// TIA Portal project "Seviye ve Sıcaklık Kontrol" (V17)

(* hardware
DEVICE "S7-1500/ET200MP station_1"  S7-1500 station
   slot 0: "Rail_0"  Rack  6ES7 590-1***0-0AA0
   slot 1: "PLC_1"  CPU 1511C-1 PN  6ES7 511-1CK00-0AB0  V2.9
      slot 3: "CPU display_1"  6ES7591-1AA00-0AA0
      slot 32768: "PROFINET interface_1"  X1
         slot 32769: "Port_1"  X1 P1
         slot 32770: "Port_2"  X1 P2
      slot 34817: "Virtual CP interface port_1"  Virtual CP interface port  Virtual CP interface port
DEVICE "HMI_1"  TP700 Comfort
   slot 0: "HMI_1"  TP700 Comfort  6AV2 124-0GC01-0AX0  17.0.0.0
   slot 1: "HMI_RT_1"  TP700 Comfort  6AV2 124-0GC01-0AX0  17.0.0.0
   slot 5: "HMI_1.IE_CP_1"  PROFINET Interface  17.0.0.0
      slot 1: "PROFINET Interface_1"  PROFINET Interface
         slot 1: "Port_1"  Port
         slot 2: "Port_2"  Port
   slot 7: "HMI_1.MPI/DP_CP_1"  MPI/DP Interface  17.0.0.0
*)

// ===== PLC "PLC_1"  CPU 1511C-1 PN =====

VAR_GLOBAL   // PLC tag table "Default tag table"
   "Otomatik Çalışma Aktif" AT %M1.0 : Bool;
   "Seviye Set Değer" AT %MD60 : Real;
   "Sıcaklık Set Değer" AT %MD40 : Real;
   "Seviye_OK" AT %M1.3 : Bool;
   "Taşma_Sensörü" AT %MD116 : Real;
   "Tag_1" AT %MD132 : DWord;
   "Anlık Seviye" AT %MD30 : DWord;
   "Anlık Sıcaklık Değeri" AT %MD46 : DWord;
   "Sistem Sıcaklık Değeri" AT %MD62 : DWord;
   "Sistem Seviye Değeri" AT %MD78 : DWord;
   "Manuel Çalışma Aktif" AT %M1.6 : Bool;
   "Sıcaklık_OK" AT %M1.1 : Bool;
   "Kullanıcıdan Alınan Zaman Değeri (Dakika)" AT %MD8 : Time;
   "Timer Zaman Değeri" AT %MD16 : Time;
   "Sistem Tamamlandı" AT %M1.2 : Bool;
   "Sistem Aşırı Sıcak" AT %M1.4 : Bool;
   "Sistem Aşırı Seviye" AT %M1.5 : Bool;
END_VAR

VAR_GLOBAL   // PLC tag table "Dijital Outputlar"
   "Pompa Motoru" AT %Q4.0 : Bool;
   "Isıtıcı" AT %Q4.1 : Bool;
   "Karıştırma Motoru" AT %Q4.2 : Bool;
   "System_OK Sesli Uyarı Sireni" AT %Q4.3 : Bool;
   "System OK Lamba" AT %Q4.4 : Bool;
   "Uyarı Kırmızı Lamba" AT %Q4.5 : Bool;
   "Uyarı Sireni" AT %Q4.6 : Bool;
   "Pompa Motoru Sürücüsü" AT %Q4.7 : Bool;
   "Karıştırma Motoru Sürücüsü" AT %Q5.0 : Bool;
END_VAR

VAR_GLOBAL   // PLC tag table "Analog Output"
   "Pompa Motoru Sürücü" AT %QW0 : Int;
   "SCR" AT %QW2 : Int;
END_VAR

VAR_GLOBAL   // PLC tag table "Dijital Inputlar"
   "Oto Start" AT %I10.0 : Bool;
   "Manuel Start Butonu" AT %I10.1 : Bool;
   "Stop Butonu" AT %I10.2 : Bool;
   "Acil Stop Butonu" AT %I10.3 : Bool;
   "Pompa Motoru Manuel Çalışma" AT %I10.4 : Bool;
   "Isıtıcı Manuel Çalışma" AT %I10.5 : Bool;
   "Karıştırma Motoru Manuel Çalıştırma Butonu" AT %I10.6 : Bool;
END_VAR

VAR_GLOBAL   // PLC tag table "Analog Inputlar"
   "Seviye Ölçer Sensörü" AT %IW0 : Int;
   "Pt100" AT %IW2 : Int;
   "Sistem Sıcaklık Sensörü" AT %IW4 : Word;
   "Taşma Sensörü" AT %IW6 : Word;
END_VAR

DATA_BLOCK "db_HMI"   // DB2
{ S7_Optimized_Access := 'TRUE' }
VERSION : 0.1
   VAR
      "Pompa Motoru Manuel Çalışma" : Bool;
      "Isıtıcı Manuel Çalışma" : Bool;
      "Karıştırma Motoru Manuel Çalıştırma" : Bool;
      "Seviye PID Manuel Çalışma" : Bool;
      "Sıcaklık PID Manuel Çalışma" : Bool;
      "HMI Oto Start" : Bool;
      "HMI Manuel Start" : Bool;
   END_VAR
BEGIN
END_DATA_BLOCK

DATA_BLOCK "db_Alarmlar"   // DB4
{ S7_Optimized_Access := 'FALSE' }
VERSION : 0.1
   VAR
      "Stop Butonuna Basıldı" : Bool;
      "Acil Stop Butonu Basılı" : Bool;
      "Sistem Aşırı Sıcak Değeri" : Bool;
      "Sistem Aşırı Seviye Değeri" : Bool;
      "Seviye Ölçer Sensörü Kablosu Koptu" : Bool;
      "Pt100 Sensörü Kablosu Koptu" : Bool;
      "Taşma Sensörü Kablosu Koptu" : Bool;
      "Sistem Sıcaklık Sensörü Kablosu Koptu" : Bool;
   END_VAR
BEGIN
END_DATA_BLOCK

// folder: System blocks/Program resources

DATA_BLOCK "Zamanlayıcı"   // DB5
{ S7_Optimized_Access := 'TRUE' }
AUTHOR : Simatic
FAMILY : IEC
NAME : IEC_TMR
VERSION : 1.0
// stored: InstanceOfName IEC_TIMER
"IEC_TIMER"
BEGIN
END_DATA_BLOCK

// folder: (top level)

FUNCTION "HMI Alarmlar" : Void   // FC1, LAD
{ S7_Optimized_Access := 'TRUE' }
VERSION : 0.1
BEGIN

REGION Network 1
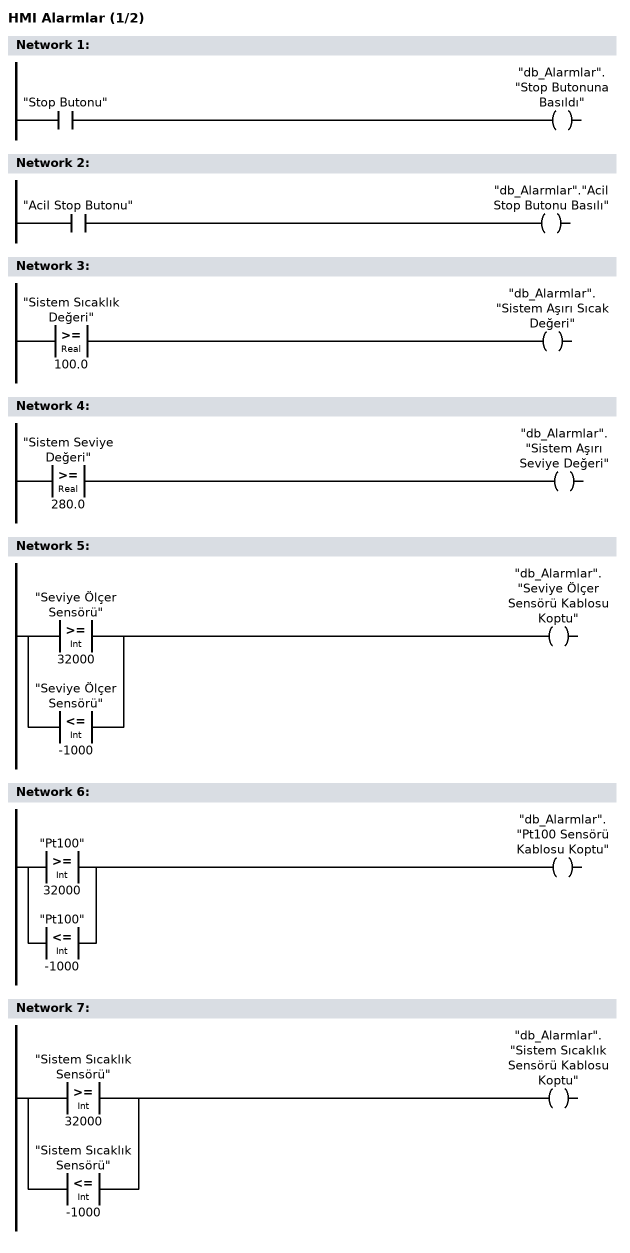
   RUNG wire#powerrail
      Contact( "Stop Butonu" )
      Coil( "db_Alarmlar"."Stop Butonuna Basıldı" )
   END_RUNG
   // the same network as SCL:
   "db_Alarmlar"."Stop Butonuna Basıldı" := "Stop Butonu";
END_REGION

REGION Network 2
   RUNG wire#powerrail
      Contact( "Acil Stop Butonu" )
      Coil( "db_Alarmlar"."Acil Stop Butonu Basılı" )
   END_RUNG
   // the same network as SCL:
   "db_Alarmlar"."Acil Stop Butonu Basılı" := "Acil Stop Butonu";
END_REGION

REGION Network 3
   RUNG wire#powerrail
      { S7_Templates := "SrcType := Real" } GE_Contact(in1 := "Sistem Sıcaklık Değeri", in2 := 100.0)
      Coil( "db_Alarmlar"."Sistem Aşırı Sıcak Değeri" )
   END_RUNG
   // the same network as SCL:
   "db_Alarmlar"."Sistem Aşırı Sıcak Değeri" := "Sistem Sıcaklık Değeri" >= 100.0;
END_REGION

REGION Network 4
   RUNG wire#powerrail
      { S7_Templates := "SrcType := Real" } GE_Contact(in1 := "Sistem Seviye Değeri", in2 := 280.0)
      Coil( "db_Alarmlar"."Sistem Aşırı Seviye Değeri" )
   END_RUNG
   // the same network as SCL:
   "db_Alarmlar"."Sistem Aşırı Seviye Değeri" := "Sistem Seviye Değeri" >= 280.0;
END_REGION

REGION Network 5
   RUNG wire#powerrail
      { S7_Templates := "SrcType := Int" } GE_Contact(in1 := "Seviye Ölçer Sensörü", in2 := 32000)
      wire#w1
      Coil( "db_Alarmlar"."Seviye Ölçer Sensörü Kablosu Koptu" )
   END_RUNG
   RUNG wire#powerrail
      { S7_Templates := "SrcType := Int" } LE_Contact(in1 := "Seviye Ölçer Sensörü", in2 := -1000)
   END_RUNG wire#w1
   // the same network as SCL:
   "db_Alarmlar"."Seviye Ölçer Sensörü Kablosu Koptu" := ("Seviye Ölçer Sensörü" >= 32000) OR ("Seviye Ölçer Sensörü" <= (-1000));
END_REGION

REGION Network 6
   RUNG wire#powerrail
      { S7_Templates := "SrcType := Int" } GE_Contact(in1 := "Pt100", in2 := 32000)
      wire#w1
      Coil( "db_Alarmlar"."Pt100 Sensörü Kablosu Koptu" )
   END_RUNG
   RUNG wire#powerrail
      { S7_Templates := "SrcType := Int" } LE_Contact(in1 := "Pt100", in2 := -1000)
   END_RUNG wire#w1
   // the same network as SCL:
   "db_Alarmlar"."Pt100 Sensörü Kablosu Koptu" := ("Pt100" >= 32000) OR ("Pt100" <= (-1000));
END_REGION

REGION Network 7
   RUNG wire#powerrail
      { S7_Templates := "SrcType := Int" } GE_Contact(in1 := "Sistem Sıcaklık Sensörü", in2 := 32000)
      wire#w1
      Coil( "db_Alarmlar"."Sistem Sıcaklık Sensörü Kablosu Koptu" )
   END_RUNG
   RUNG wire#powerrail
      { S7_Templates := "SrcType := Int" } LE_Contact(in1 := "Sistem Sıcaklık Sensörü", in2 := -1000)
   END_RUNG wire#w1
   // the same network as SCL:
   "db_Alarmlar"."Sistem Sıcaklık Sensörü Kablosu Koptu" := ("Sistem Sıcaklık Sensörü" >= 32000) OR ("Sistem Sıcaklık Sensörü" <= (-1000));
END_REGION

REGION Network 8
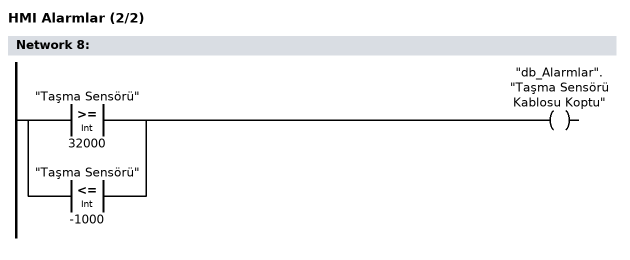
   RUNG wire#powerrail
      { S7_Templates := "SrcType := Int" } GE_Contact(in1 := "Taşma Sensörü", in2 := 32000)
      wire#w1
      Coil( "db_Alarmlar"."Taşma Sensörü Kablosu Koptu" )
   END_RUNG
   RUNG wire#powerrail
      { S7_Templates := "SrcType := Int" } LE_Contact(in1 := "Taşma Sensörü", in2 := -1000)
   END_RUNG wire#w1
   // the same network as SCL:
   "db_Alarmlar"."Taşma Sensörü Kablosu Koptu" := ("Taşma Sensörü" >= 32000) OR ("Taşma Sensörü" <= (-1000));
END_REGION
END_FUNCTION

FUNCTION "Manuel Çalışma" : Void   // FC2, LAD
{ S7_Optimized_Access := 'TRUE' }
VERSION : 0.1
BEGIN

REGION Network 1: Manuel Çalışma Modu
   // Manuel Start ile Merker biti aktif edilir.
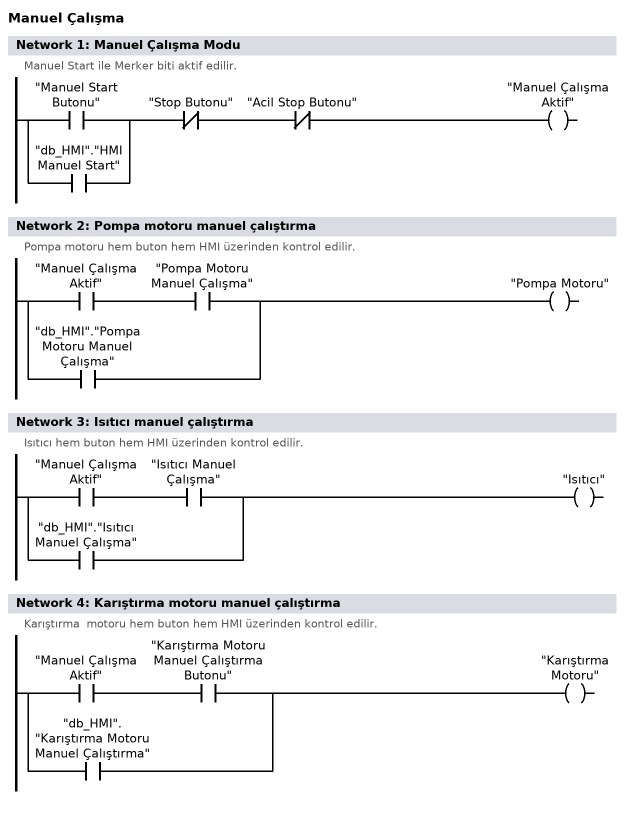
   RUNG wire#powerrail
      Contact( "Manuel Start Butonu" )
      wire#w1
      I_Contact( "Stop Butonu" )
      I_Contact( "Acil Stop Butonu" )
      Coil( "Manuel Çalışma Aktif" )
   END_RUNG
   RUNG wire#powerrail
      Contact( "db_HMI"."HMI Manuel Start" )
   END_RUNG wire#w1
   // the same network as SCL:
   "Manuel Çalışma Aktif" := ("Manuel Start Butonu" OR "db_HMI"."HMI Manuel Start") AND NOT "Stop Butonu" AND NOT "Acil Stop Butonu";
END_REGION

REGION Network 2: Pompa motoru manuel çalıştırma
   // Pompa motoru hem buton hem HMI üzerinden kontrol edilir.
   RUNG wire#powerrail
      Contact( "Manuel Çalışma Aktif" )
      Contact( "Pompa Motoru Manuel Çalışma" )
      wire#w1
      Coil( "Pompa Motoru" )
   END_RUNG
   RUNG wire#powerrail
      Contact( "db_HMI"."Pompa Motoru Manuel Çalışma" )
   END_RUNG wire#w1
   // the same network as SCL:
   "Pompa Motoru" := ("Manuel Çalışma Aktif" AND "Pompa Motoru Manuel Çalışma") OR "db_HMI"."Pompa Motoru Manuel Çalışma";
END_REGION

REGION Network 3: Isıtıcı manuel çalıştırma
   // Isıtıcı hem buton hem HMI üzerinden kontrol edilir.
   RUNG wire#powerrail
      Contact( "Manuel Çalışma Aktif" )
      Contact( "Isıtıcı Manuel Çalışma" )
      wire#w1
      Coil( "Isıtıcı" )
   END_RUNG
   RUNG wire#powerrail
      Contact( "db_HMI"."Isıtıcı Manuel Çalışma" )
   END_RUNG wire#w1
   // the same network as SCL:
   "Isıtıcı" := ("Manuel Çalışma Aktif" AND "Isıtıcı Manuel Çalışma") OR "db_HMI"."Isıtıcı Manuel Çalışma";
END_REGION

REGION Network 4: Karıştırma motoru manuel çalıştırma
   // Karıştırma  motoru hem buton hem HMI üzerinden kontrol edilir.
   RUNG wire#powerrail
      Contact( "Manuel Çalışma Aktif" )
      Contact( "Karıştırma Motoru Manuel Çalıştırma Butonu" )
      wire#w1
      Coil( "Karıştırma Motoru" )
   END_RUNG
   RUNG wire#powerrail
      Contact( "db_HMI"."Karıştırma Motoru Manuel Çalıştırma" )
   END_RUNG wire#w1
   // the same network as SCL:
   "Karıştırma Motoru" := ("Manuel Çalışma Aktif" AND "Karıştırma Motoru Manuel Çalıştırma Butonu") OR "db_HMI"."Karıştırma Motoru Manuel Çalıştırma";
END_REGION
END_FUNCTION

FUNCTION "Otomatik Çalışma" : Void   // FC3, LAD
{ S7_Optimized_Access := 'TRUE' }
VERSION : 0.1
BEGIN

REGION Network 1: Başlangıç
   // Start butonuna basarak sistemi aktif ederiz. Sistem aktif bilgisini merker bitiyle bağlayıp diğer adımlarda rahatlıkla kullanılır.
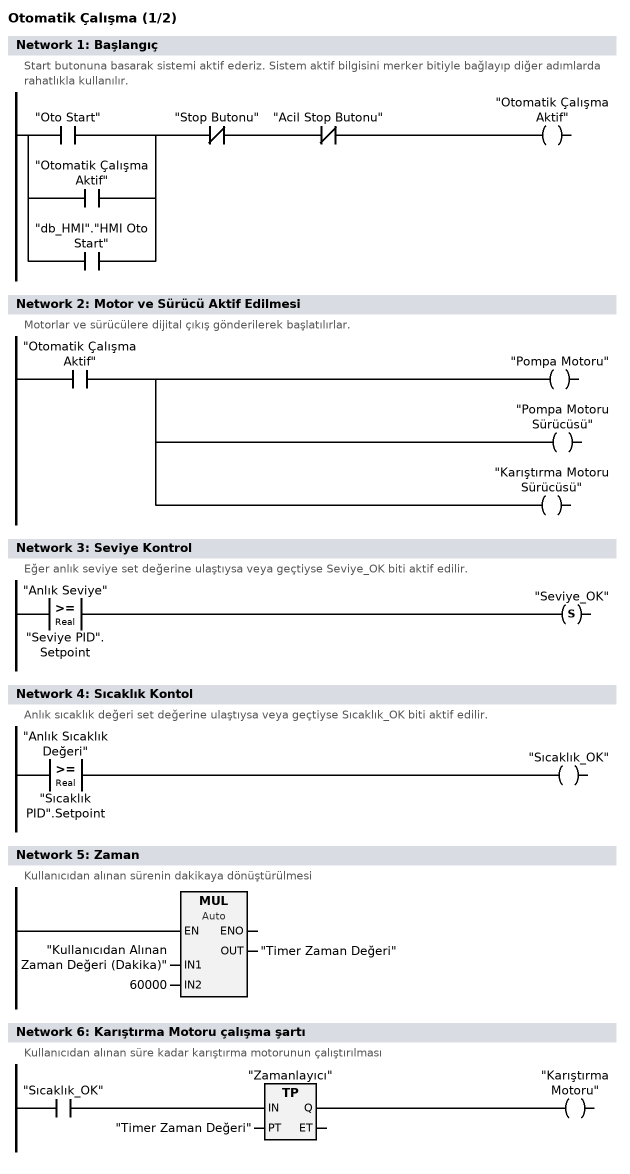
   RUNG wire#powerrail
      Contact( "Oto Start" )
      wire#w1
      I_Contact( "Stop Butonu" )
      I_Contact( "Acil Stop Butonu" )
      Coil( "Otomatik Çalışma Aktif" )
   END_RUNG
   RUNG wire#powerrail
      Contact( "Otomatik Çalışma Aktif" )
   END_RUNG wire#w1
   RUNG wire#powerrail
      Contact( "db_HMI"."HMI Oto Start" )
   END_RUNG wire#w1
   // the same network as SCL:
   "Otomatik Çalışma Aktif" := ("Oto Start" OR "Otomatik Çalışma Aktif" OR "db_HMI"."HMI Oto Start") AND NOT "Stop Butonu" AND NOT "Acil Stop Butonu";
END_REGION

REGION Network 2: Motor ve Sürücü Aktif Edilmesi
   // Motorlar ve sürücülere dijital çıkış gönderilerek başlatılırlar.
   RUNG wire#powerrail
      Contact( "Otomatik Çalışma Aktif" )
      wire#w1
      Coil( "Pompa Motoru" )
   END_RUNG
   RUNG wire#w1
      Coil( "Pompa Motoru Sürücüsü" )
   END_RUNG
   RUNG wire#w1
      Coil( "Karıştırma Motoru Sürücüsü" )
   END_RUNG
   // the same network as SCL:
   "Pompa Motoru" := "Otomatik Çalışma Aktif";
   "Pompa Motoru Sürücüsü" := "Otomatik Çalışma Aktif";
   "Karıştırma Motoru Sürücüsü" := "Otomatik Çalışma Aktif";
END_REGION

REGION Network 3: Seviye Kontrol
   // Eğer anlık seviye set değerine ulaştıysa veya geçtiyse Seviye_OK biti aktif edilir.
   RUNG wire#powerrail
      { S7_Templates := "SrcType := Real" } GE_Contact(in1 := "Anlık Seviye", in2 := "Seviye PID".Setpoint)
      S_Coil( "Seviye_OK" )
   END_RUNG
   // the same network as SCL:
   IF "Anlık Seviye" >= "Seviye PID".Setpoint THEN "Seviye_OK" := TRUE; END_IF;
END_REGION

REGION Network 4: Sıcaklık Kontol
   // Anlık sıcaklık değeri set değerine ulaştıysa veya geçtiyse Sıcaklık_OK biti aktif edilir.
   RUNG wire#powerrail
      { S7_Templates := "SrcType := Real" } GE_Contact(in1 := "Anlık Sıcaklık Değeri", in2 := "Sıcaklık PID".Setpoint)
      Coil( "Sıcaklık_OK" )
   END_RUNG
   // the same network as SCL:
   "Sıcaklık_OK" := "Anlık Sıcaklık Değeri" >= "Sıcaklık PID".Setpoint;
END_REGION

REGION Network 5: Zaman
   // Kullanıcıdan alınan sürenin dakikaya dönüştürülmesi
   RUNG wire#powerrail
      Mul(in1 := "Kullanıcıdan Alınan Zaman Değeri (Dakika)", in2 := 60000, out => "Timer Zaman Değeri")
   END_RUNG
   // the same network as SCL:
   "Timer Zaman Değeri" := "Kullanıcıdan Alınan Zaman Değeri (Dakika)" * 60000;
END_REGION

REGION Network 6: Karıştırma Motoru çalışma şartı
   // Kullanıcıdan alınan süre kadar karıştırma motorunun çalıştırılması
   "Zamanlayıcı".TP(IN := "Sıcaklık_OK", PT := "Timer Zaman Değeri");
   "Karıştırma Motoru" := "Zamanlayıcı".Q;
END_REGION

REGION Network 7: Sistemin tamamlanması
   // Seviye set değerine ulaştıysa, Sıcaklık set değerine ulaştıysa ve karıştıma motoru istenilen zaman aralığında çalıştıysa sistem tamamlandı demektir.
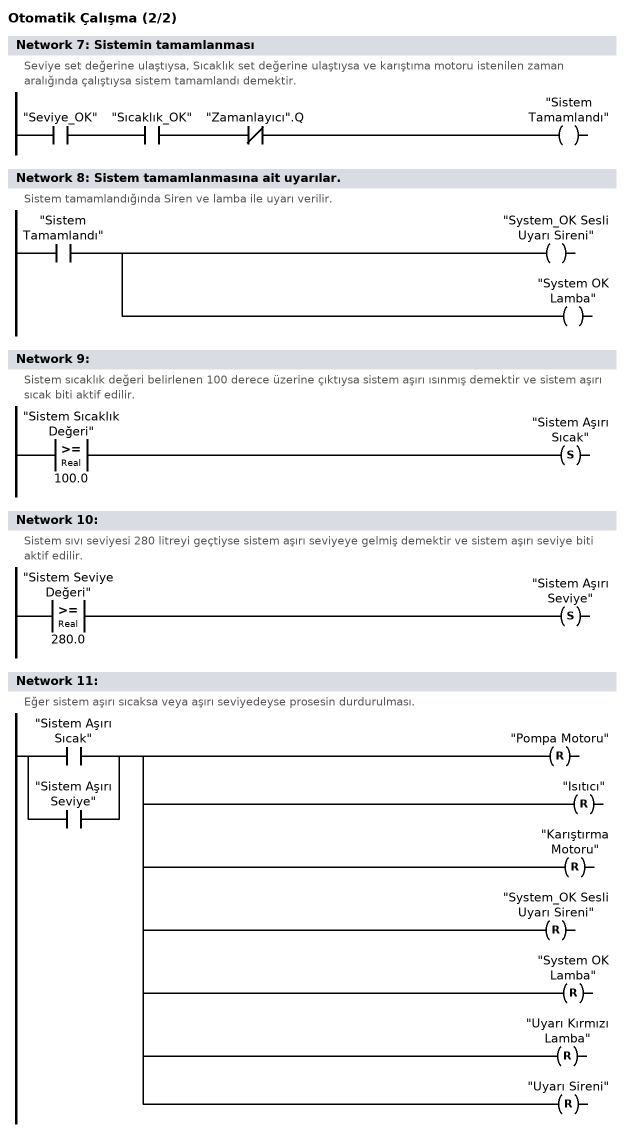
   RUNG wire#powerrail
      Contact( "Seviye_OK" )
      Contact( "Sıcaklık_OK" )
      I_Contact( "Zamanlayıcı".Q )
      Coil( "Sistem Tamamlandı" )
   END_RUNG
   // the same network as SCL:
   "Sistem Tamamlandı" := "Seviye_OK" AND "Sıcaklık_OK" AND NOT "Zamanlayıcı".Q;
END_REGION

REGION Network 8: Sistem tamamlanmasına ait uyarılar.
   // Sistem tamamlandığında Siren ve lamba ile uyarı verilir.
   RUNG wire#powerrail
      Contact( "Sistem Tamamlandı" )
      wire#w1
      Coil( "System_OK Sesli Uyarı Sireni" )
   END_RUNG
   RUNG wire#w1
      Coil( "System OK Lamba" )
   END_RUNG
   // the same network as SCL:
   "System_OK Sesli Uyarı Sireni" := "Sistem Tamamlandı";
   "System OK Lamba" := "Sistem Tamamlandı";
END_REGION

REGION Network 9
   // Sistem sıcaklık değeri belirlenen 100 derece üzerine çıktıysa sistem aşırı ısınmış demektir ve sistem aşırı sıcak biti aktif edilir.
   RUNG wire#powerrail
      { S7_Templates := "SrcType := Real" } GE_Contact(in1 := "Sistem Sıcaklık Değeri", in2 := 100.0)
      S_Coil( "Sistem Aşırı Sıcak" )
   END_RUNG
   // the same network as SCL:
   IF "Sistem Sıcaklık Değeri" >= 100.0 THEN "Sistem Aşırı Sıcak" := TRUE; END_IF;
END_REGION

REGION Network 10
   // Sistem sıvı seviyesi 280 litreyi geçtiyse sistem aşırı seviyeye gelmiş demektir ve sistem aşırı seviye biti aktif edilir.
   RUNG wire#powerrail
      { S7_Templates := "SrcType := Real" } GE_Contact(in1 := "Sistem Seviye Değeri", in2 := 280.0)
      S_Coil( "Sistem Aşırı Seviye" )
   END_RUNG
   // the same network as SCL:
   IF "Sistem Seviye Değeri" >= 280.0 THEN "Sistem Aşırı Seviye" := TRUE; END_IF;
END_REGION

REGION Network 11
   // Eğer sistem aşırı sıcaksa veya aşırı seviyedeyse prosesin durdurulması.
   RUNG wire#powerrail
      Contact( "Sistem Aşırı Sıcak" )
      wire#w1
      R_Coil( "Pompa Motoru" )
   END_RUNG
   RUNG wire#powerrail
      Contact( "Sistem Aşırı Seviye" )
   END_RUNG wire#w1
   RUNG wire#w1
      R_Coil( "Isıtıcı" )
   END_RUNG
   RUNG wire#w1
      R_Coil( "Karıştırma Motoru" )
   END_RUNG
   RUNG wire#w1
      R_Coil( "System_OK Sesli Uyarı Sireni" )
   END_RUNG
   RUNG wire#w1
      R_Coil( "System OK Lamba" )
   END_RUNG
   RUNG wire#w1
      R_Coil( "Uyarı Kırmızı Lamba" )
   END_RUNG
   RUNG wire#w1
      R_Coil( "Uyarı Sireni" )
   END_RUNG
   // the same network as SCL:
   IF "Sistem Aşırı Sıcak" OR "Sistem Aşırı Seviye" THEN
       "Pompa Motoru" := FALSE;
       "Isıtıcı" := FALSE;
       "Karıştırma Motoru" := FALSE;
       "System_OK Sesli Uyarı Sireni" := FALSE;
       "System OK Lamba" := FALSE;
       "Uyarı Kırmızı Lamba" := FALSE;
       "Uyarı Sireni" := FALSE;
   END_IF;
END_REGION
END_FUNCTION

ORGANIZATION_BLOCK "Main"   // OB1, LAD, ProgramCycle
TITLE = "Main Program Sweep (Cycle)"
{ S7_Optimized_Access := 'TRUE' }
VERSION : 0.1
   VAR_INPUT
      Initial_Call : Bool;   // Initial call of this OB
      Remanence : Bool;   // =True, if remanent data are available
   END_VAR
   VAR_TEMP
      NORMX_Out : Real;
      NORMX_Out_1 : Real;
      NORMX_Out_2 : Real;
      NORMX_Out_3 : Real;
   END_VAR
BEGIN

REGION Network 1: Seviye Ölçer Sensörü Normalizasyon ve Skala İşlemi
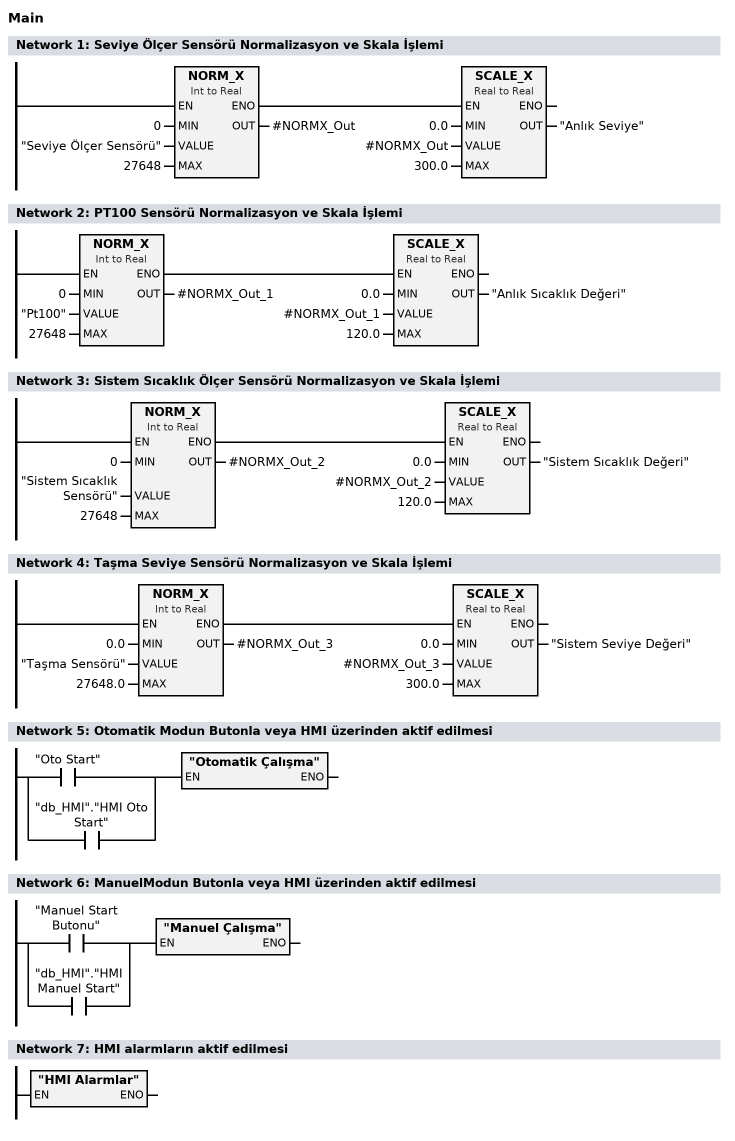
   RUNG wire#powerrail
      { S7_Templates := "[SrcType := Int, DestType := Real]" } Normalize(min := 0, value := "Seviye Ölçer Sensörü", max := 27648, out => #NORMX_Out)
      { S7_Templates := "[SrcType := Real, DestType := Real]" } Scale(min := 0.0, value := #NORMX_Out, max := 300.0, out => "Anlık Seviye")
   END_RUNG
   // the same network as SCL:
   #NORMX_Out := NORM_X(MIN := 0, VALUE := "Seviye Ölçer Sensörü", MAX := 27648);
   "Anlık Seviye" := SCALE_X(MIN := 0.0, VALUE := #NORMX_Out, MAX := 300.0);
END_REGION

REGION Network 2: PT100 Sensörü Normalizasyon ve Skala İşlemi
   RUNG wire#powerrail
      { S7_Templates := "[SrcType := Int, DestType := Real]" } Normalize(min := 0, value := "Pt100", max := 27648, out => #NORMX_Out_1)
      { S7_Templates := "[SrcType := Real, DestType := Real]" } Scale(min := 0.0, value := #NORMX_Out_1, max := 120.0, out => "Anlık Sıcaklık Değeri")
   END_RUNG
   // the same network as SCL:
   #NORMX_Out_1 := NORM_X(MIN := 0, VALUE := "Pt100", MAX := 27648);
   "Anlık Sıcaklık Değeri" := SCALE_X(MIN := 0.0, VALUE := #NORMX_Out_1, MAX := 120.0);
END_REGION

REGION Network 3: Sistem Sıcaklık Ölçer Sensörü Normalizasyon ve Skala İşlemi
   RUNG wire#powerrail
      { S7_Templates := "[SrcType := Int, DestType := Real]" } Normalize(min := 0, value := "Sistem Sıcaklık Sensörü", max := 27648, out => #NORMX_Out_2)
      { S7_Templates := "[SrcType := Real, DestType := Real]" } Scale(min := 0.0, value := #NORMX_Out_2, max := 120.0, out => "Sistem Sıcaklık Değeri")
   END_RUNG
   // the same network as SCL:
   #NORMX_Out_2 := NORM_X(MIN := 0, VALUE := "Sistem Sıcaklık Sensörü", MAX := 27648);
   "Sistem Sıcaklık Değeri" := SCALE_X(MIN := 0.0, VALUE := #NORMX_Out_2, MAX := 120.0);
END_REGION

REGION Network 4: Taşma Seviye Sensörü Normalizasyon ve Skala İşlemi
   RUNG wire#powerrail
      { S7_Templates := "[SrcType := Int, DestType := Real]" } Normalize(min := 0.0, value := "Taşma Sensörü", max := 27648.0, out => #NORMX_Out_3)
      { S7_Templates := "[SrcType := Real, DestType := Real]" } Scale(min := 0.0, value := #NORMX_Out_3, max := 300.0, out => "Sistem Seviye Değeri")
   END_RUNG
   // the same network as SCL:
   #NORMX_Out_3 := NORM_X(MIN := 0.0, VALUE := "Taşma Sensörü", MAX := 27648.0);
   "Sistem Seviye Değeri" := SCALE_X(MIN := 0.0, VALUE := #NORMX_Out_3, MAX := 300.0);
END_REGION

REGION Network 5: Otomatik Modun Butonla veya HMI üzerinden aktif edilmesi
   RUNG wire#powerrail
      Contact( "Oto Start" )
      wire#w1
      "Otomatik Çalışma"()
   END_RUNG
   RUNG wire#powerrail
      Contact( "db_HMI"."HMI Oto Start" )
   END_RUNG wire#w1
   // the same network as SCL:
   IF "Oto Start" OR "db_HMI"."HMI Oto Start" THEN "Otomatik Çalışma"(); END_IF;
END_REGION

REGION Network 6: ManuelModun Butonla veya HMI üzerinden aktif edilmesi
   RUNG wire#powerrail
      Contact( "Manuel Start Butonu" )
      wire#w1
      "Manuel Çalışma"()
   END_RUNG
   RUNG wire#powerrail
      Contact( "db_HMI"."HMI Manuel Start" )
   END_RUNG wire#w1
   // the same network as SCL:
   IF "Manuel Start Butonu" OR "db_HMI"."HMI Manuel Start" THEN "Manuel Çalışma"(); END_IF;
END_REGION

REGION Network 7: HMI alarmların aktif edilmesi
   RUNG wire#powerrail
      "HMI Alarmlar"()
   END_RUNG
   // the same network as SCL:
   "HMI Alarmlar"();
END_REGION
END_ORGANIZATION_BLOCK

ORGANIZATION_BLOCK "Seviye PID Kontrol"   // OB30, LAD, CyclicInterrupt
{ S7_Optimized_Access := 'TRUE' }
VERSION : 0.1
   VAR_INPUT
      Initial_Call : Bool;   // Initial call of this OB
      Event_Count : Int;   // Events discarded
   END_VAR
BEGIN

REGION Network 1: Seviye PID bloğunun aktif edilmesi
   // Hem otomatik hem manuel modda aktif edilebilir. Setpoint kısmına hafıza bitiatayarak HMI üzerinden değer girilebilir. Input_PER kısmını analog input girilir. Output_PER kısmına analog çıkış atanır. Seviye kontrolü için seviye bilgisi veren, analog seviye ölçer sensörünü Input_PER kısmına girip seviye değeri alınır. Daha sonra çıkışa motoru hız kontrollü çalıştırmak için sürücü atanır. Sürücü frekans artırıp azaltarak sürücüyü hız kontrolle çalıştırır.
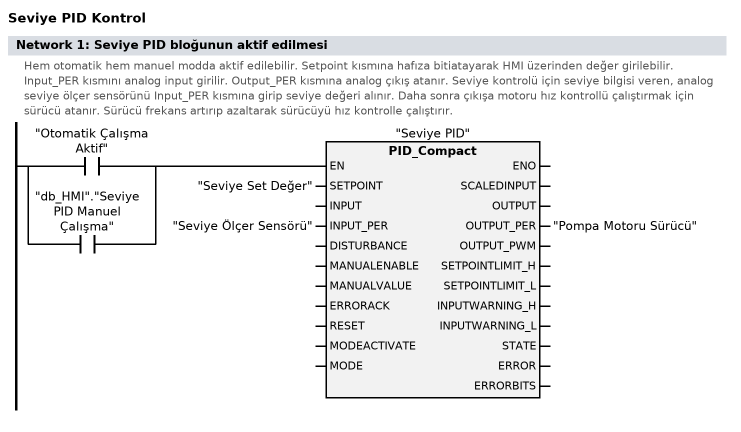
   IF "Otomatik Çalışma Aktif" OR "db_HMI"."Seviye PID Manuel Çalışma" THEN
       "Seviye PID"(Setpoint := "Seviye Set Değer",   // PID_Compact
                    Input_PER := "Seviye Ölçer Sensörü",
                    Output_PER => "Pompa Motoru Sürücü");
   END_IF;
END_REGION
END_ORGANIZATION_BLOCK

ORGANIZATION_BLOCK "Sıcaklık PID Kontrol"   // OB31, LAD, CyclicInterrupt
{ S7_Optimized_Access := 'TRUE' }
VERSION : 0.1
   VAR_INPUT
      Initial_Call : Bool;   // Initial call of this OB
      Event_Count : Int;   // Events discarded
   END_VAR
BEGIN

REGION Network 1: Sıcaklık PID Bloğunun Aktif Edilmesi
   // Setpoint kısmına hafıza bitiatayarak HMI üzerinden değer girilebilir. Input_PER kısmını analog input girilir. Output_PER kısmına analog çıkış atanır. Sıcalık kontrolü için sıcaklık bilgisi veren, pt100 sensörünü Input_PER kısmına girip seviye değeri alınır. Daha sonra çıkışa ısıtıcıyı kademeli olarak  çalıştırmak için scr cihazı atanır.
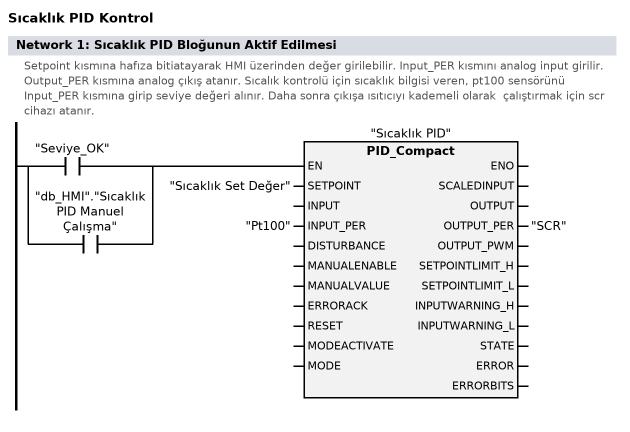
   IF "Seviye_OK" OR "db_HMI"."Sıcaklık PID Manuel Çalışma" THEN
       "Sıcaklık PID"(Setpoint := "Sıcaklık Set Değer", Input_PER := "Pt100", Output_PER => "SCR");   // PID_Compact
   END_IF;
END_REGION
END_ORGANIZATION_BLOCK

(* ===== HMI "HMI_RT_1" =====
system functions are stored by id; their names below are inferred from use
connection "HMI_Connection_1": ETHERNET, S7_1500_OMS

HMI tags "Default tag table"
   "Tag_ScreenNumber" : UInt, internal
   "db_HMI_HMI Oto Start" : Bool = PLC db_HMI."HMI Oto Start", 1 s
   "db_HMI_HMI Manuel Start" : Bool = PLC db_HMI."HMI Manuel Start", 1 s
   "Sistem Seviye Değeri" : DWord = PLC "Sistem Seviye Değeri" AT %MD78, 1 s
   "Sistem Sıcaklık Değeri" : DWord = PLC "Sistem Sıcaklık Değeri" AT %MD62, 1 s
   "Kullanıcıdan Alınan Zaman Değeri (Dakika)" : Time = PLC "Kullanıcıdan Alınan Zaman Değeri (Dakika)" AT %MD8, 1 s
   "db_HMI_Pompa Motoru Manuel Çalışma" : Bool = PLC db_HMI."Pompa Motoru Manuel Çalışma", 1 s
   "db_HMI_Isıtıcı Manuel Çalışma" : Bool = PLC db_HMI."Isıtıcı Manuel Çalışma", 1 s
   "db_HMI_Karıştırma Motoru Manuel Çalıştırma" : Bool = PLC db_HMI."Karıştırma Motoru Manuel Çalıştırma", 1 s
   "Pompa Motoru" : Bool = PLC "Pompa Motoru" AT %Q4.0, 1 s
   "Isıtıcı" : Bool = PLC Isıtıcı AT %Q4.1, 1 s
   "Karıştırma Motoru" : Bool = PLC "Karıştırma Motoru" AT %Q4.2, 1 s
   "Seviye Set Değer" : Real = PLC "Seviye Set Değer" AT %MD60, 1 s
   "Anlık Seviye" : DWord = PLC "Anlık Seviye" AT %MD30, 1 s
   "Seviye PID_Retain_CtrlParams_Ti" : Real = PLC "Seviye PID".Retain.CtrlParams.Ti, 1 s
   "Seviye PID_Retain_CtrlParams_Gain" : Real = PLC "Seviye PID".Retain.CtrlParams.Gain, 1 s
   "Seviye PID_Retain_CtrlParams_Td" : Real = PLC "Seviye PID".Retain.CtrlParams.Td, 1 s
   "Anlık Sıcaklık Değeri" : DWord = PLC "Anlık Sıcaklık Değeri" AT %MD46, 1 s
   "Sıcaklık Set Değer" : Real = PLC "Sıcaklık Set Değer" AT %MD40, 1 s
   "Sıcaklık PID_Retain_CtrlParams_Gain" : Real = PLC "Sıcaklık PID".Retain.CtrlParams.Gain, 1 s
   "Sıcaklık PID_Retain_CtrlParams_Ti" : Real = PLC "Sıcaklık PID".Retain.CtrlParams.Ti, 1 s
   "Sıcaklık PID_Retain_CtrlParams_Td" : Real = PLC "Sıcaklık PID".Retain.CtrlParams.Td, 1 s
   "Alarm" : UInt AT %DB1.DBW0, 1 s
   "Seviye PID_ScaledInput" : Real = PLC "Seviye PID".ScaledInput, 1 s
   "Sıcaklık PID_ScaledInput" : Real = PLC "Sıcaklık PID".ScaledInput, 1 s
   "Pt100" : Int = PLC Pt100 AT %IW2, 1 s

discrete alarms
   8: 'Sistem Sıcaklık Sensörü Kablosu Koptu', class Errors, trigger "Alarm" bit 15
   7: 'Taşma Sensörü Kablosu Koptu', class Errors, trigger "Alarm" bit 14
   6: 'Pt100 Sensörü Kablosu Koptu', class Errors, trigger "Alarm" bit 13
   5: 'Seviye Ölçer Sensörü Kablosu Koptu', class Errors, trigger "Alarm" bit 12
   4: 'Sistem Aşırı Seviye Değeri', class Errors, trigger "Alarm" bit 11
   3: 'Sistem Aşırı Sıcak Değeri', class Errors, trigger "Alarm" bit 10
   2: 'Acil Stop Butonu Basılı', class Errors, trigger "Alarm" bit 9
   1: 'Stop Butonuna Basıldı', class Errors, trigger "Alarm" bit 8

graphic list "Karıştırma Motoru": 0 'Graphic_4'; 1 'Graphic_9'

graphic list "Pompa Motoru": 0 'Graphic_1'; 1 'Graphic_8'

graphic list "Isıtıcı": 0 'Graphic_6'; 1 'Graphic_7'

recipe "Sıcaklık PID Parametleri": PID Gain <- "Sıcaklık PID_Retain_CtrlParams_Gain", PID Ti <- "Sıcaklık PID_Retain_CtrlParams_Ti", PID Td <- "Sıcaklık PID_Retain_CtrlParams_Td"

recipe "Seviye PID Parametreleri": PID Gain <- "Seviye PID_Retain_CtrlParams_Gain", PID Ti <- "Seviye PID_Retain_CtrlParams_Ti", PID Td <- "Seviye PID_Retain_CtrlParams_Td"

screen "Ana Sayfa" 800x420, template "Template_1"
   on GenerateScreen: SetTag("Tag_ScreenNumber", 1)
   Button "Button_1" at 1,2 size 106x32; TextOff 'Otomatik Mod'
      on Press: InvertBit("db_HMI_HMI Oto Start"); ResetBit("db_HMI_HMI Manuel Start")
      Appearance <- "db_HMI_HMI Oto Start"
   Button "Button_2" at 0,33 size 106x32; TextOff 'Manuel Mod'
      on Press: InvertBit("db_HMI_HMI Manuel Start"); ResetBit("db_HMI_HMI Oto Start")
      Appearance <- "db_HMI_HMI Manuel Start"
   IOField "I/O field_1" at 134,99 size 96x32; FormatPattern 999
      ProcessValue <- "Sistem Seviye Değeri"
   IOField "I/O field_2" at 134,143 size 96x32; FormatPattern 999
      ProcessValue <- "Sistem Sıcaklık Değeri"
   TextField "Text field_1" at 10,101 size 116x20; Text 'Taşma Sensörü'
   TextField "Text field_2" at 11,134 size 114x36; Text 'Sistem Sıcaklık Sensörü'
   TextField "Text field_3" at 3,189 size 140x36; Text 'Karıştırma Motoru Çalıştırma Süresi'
   GraphicView "Graphic view_2" at 506,61 size 195x272; Picture "Graphic_3"
   Button "Button_3" at 443,258 size 77x84; TextOff 'Text'; PictureList "Pompa Motoru"
      ProcessValue <- "Pompa Motoru"
   Button "Button_4" at 696,258 size 77x84; TextOff 'Text'; PictureList "Isıtıcı"
      ProcessValue <- "Isıtıcı"
   Button "Button_5" at 574,94 size 57x164; TextOff 'Text'; PictureList "Karıştırma Motoru"
      ProcessValue <- "Karıştırma Motoru"
   Button "Button_6" at 428,342 size 104x32; TextOff 'Pompa Motoru'
      on Press: InvertBit("db_HMI_Pompa Motoru Manuel Çalışma")
   Button "Button_7" at 683,342 size 104x32; TextOff 'Isıtıcı'
      on Press: InvertBit("db_HMI_Isıtıcı Manuel Çalışma")
   Button "Button_8" at 547,258 size 117x32; TextOff 'Karıştırma Motoru'
      on Press: InvertBit("db_HMI_Karıştırma Motoru Manuel Çalıştırma")
   Button "Button_9" at 1,388 size 96x32; TextOff 'Seviye PID'
      on Click: ActivateScreen("Seviye PID", 0)
   Button "Button_10" at 96,388 size 96x32; TextOff 'Sıcaklık PID'
      on Click: ActivateScreen("Sıcaklık PID", 0)
   Button "Button_11" at 190,388 size 108x32; TextOff 'Reçete Sayfası'
      on Click: ActivateScreen("Reçete", 0)
   IOField "I/O field_3" at 131,194 size 96x32; FormatPattern 999999
      ProcessValue <- "Kullanıcıdan Alınan Zaman Değeri (Dakika)"
   Button "Button_12" at 295,388 size 96x32; TextOff 'Trend Grafiği'
      on Click: ActivateScreen("Trend Grafiği", 0)

screen "Seviye PID" 800x420
   TextField "Text field_1" at 141,101 size 153x20; Text 'Tank Sıvı Set Değeri'
   TextField "Text field_2" at 124,134 size 187x20; Text 'Tank Seviye Anlık Değeri'
   TextField "Text field_3" at 174,210 size 66x20; Text 'PID Gain'
   GraphicView "Graphic view_2" at 446,59 size 195x272; Picture "Graphic_3"
   IOField "I/O field_1" at 311,99 size 96x32
      ProcessValue <- "Seviye Set Değer"
   IOField "I/O field_2" at 311,134 size 96x32; FormatPattern 999999999.999
      ProcessValue <- "Seviye PID_ScaledInput"
   TextField "Text field_4" at 183,239 size 47x20; Text 'PID Ti'
   TextField "Text field_5" at 181,268 size 52x20; Text 'PID Td'
   IOField "I/O field_3" at 300,208 size 96x32
      ProcessValue <- "Seviye PID_Retain_CtrlParams_Gain"
   IOField "I/O field_4" at 300,244 size 96x32
      ProcessValue <- "Seviye PID_Retain_CtrlParams_Ti"
   IOField "I/O field_5" at 300,280 size 96x32
      ProcessValue <- "Seviye PID_Retain_CtrlParams_Td"
   TextField "Text field_6" at 216,60 size 111x23; Text 'PID Kontrol'
   TextField "Text field_7" at 200,177 size 171x23; Text 'PID Parametreleri'
   Button "Button_1" at 0,388 size 96x32; TextOff 'Ana Sayfa'
      on Click: ActivateScreen("Ana Sayfa", 0)
   Button "Button_11" at 191,388 size 108x32; TextOff 'Reçete Sayfası'
      on Click: ActivateScreen("Reçete", 0)
   Button "Button_10" at 96,388 size 96x32; TextOff 'Sıcaklık PID'
      on Click: ActivateScreen("Sıcaklık PID", 0)
   Button "Button_12" at 295,388 size 96x32; TextOff 'Trend Grafiği'
      on Click: ActivateScreen("Trend Grafiği", 0)

screen "Reçete" 800x420
   RecipeView "Recipe view_1" at 0,0 size 799x390; RecipeNameCaption 'Reçete Adı'; DataRecordNameCaption 'Programlar'; EntryNameCaption 'Değer Girilicekler'; ValueCaption 'Değerler'; Authorization "User administration"
   Button "Button_1" at 0,388 size 96x32; TextOff 'Ana Sayfa'
      on Click: ActivateScreen("Ana Sayfa", 0)
   Button "Button_10" at 96,388 size 96x32; TextOff 'Sıcaklık PID'
      on Click: ActivateScreen("Sıcaklık PID", 0)
   Button "Button_9" at 192,388 size 96x32; TextOff 'Seviye PID'
      on Click: ActivateScreen("Seviye PID", 0)
   Button "Button_12" at 287,388 size 96x32; TextOff 'Trend Grafiği'
      on Click: ActivateScreen("Trend Grafiği", 0)

screen "Sıcaklık PID" 800x420
   GraphicView "Graphic view_2" at 446,59 size 195x272; Picture "Graphic_3"
   TextField "Text field_1" at 135,94 size 130x36; Text 'Tank Sıvı Sıcaklık Set Değeri'
   TextField "Text field_2" at 135,134 size 130x36; Text 'Tank Sıvı Sıcaklık Anlık Değeri'
   TextField "Text field_3" at 179,210 size 66x20; Text 'PID Gain'
   TextField "Text field_4" at 188,247 size 47x20; Text 'PID Ti'
   TextField "Text field_5" at 186,286 size 52x20; Text 'PID Td'
   TextField "Text field_6" at 156,60 size 111x23; Text 'PID Kontrol'
   TextField "Text field_7" at 126,177 size 171x23; Text 'PID Parametreleri'
   IOField "I/O field_1" at 288,95 size 96x32
      ProcessValue <- "Sıcaklık Set Değer"
   IOField "I/O field_2" at 288,130 size 96x32; FormatPattern 999999999.999
      ProcessValue <- "Sıcaklık PID_ScaledInput"
   IOField "I/O field_3" at 288,204 size 96x32
      ProcessValue <- "Sıcaklık PID_Retain_CtrlParams_Gain"
   IOField "I/O field_4" at 288,239 size 96x32
      ProcessValue <- "Sıcaklık PID_Retain_CtrlParams_Ti"
   IOField "I/O field_5" at 288,279 size 96x32
      ProcessValue <- "Sıcaklık PID_Retain_CtrlParams_Td"
   Button "Button_1" at 0,388 size 96x32; TextOff 'Ana Sayfa'
      on Click: ActivateScreen("Ana Sayfa", 0)
   Button "Button_9" at 96,388 size 96x32; TextOff 'Seviye PID'
      on Click: ActivateScreen("Seviye PID", 0)
   Button "Button_11" at 191,388 size 108x32; TextOff 'Reçete Sayfası'
      on Click: ActivateScreen("Reçete", 0)
   Button "Button_12" at 295,388 size 96x32; TextOff 'Trend Grafiği'
      on Click: ActivateScreen("Trend Grafiği", 0)

screen "Trend Grafiği" 800x420
   TrendView "Trend view_1" at 1,28 size 799x361
   Button "Button_1" at 0,388 size 96x32; TextOff 'Ana Sayfa'
      on Click: ActivateScreen("Ana Sayfa", 0)
   Button "Button_10" at 96,388 size 96x32; TextOff 'Sıcaklık PID'
      on Click: ActivateScreen("Sıcaklık PID", 0)
   Button "Button_9" at 192,388 size 96x32; TextOff 'Seviye PID'
      on Click: ActivateScreen("Seviye PID", 0)
   Button "Button_11" at 287,388 size 108x32; TextOff 'Reçete Sayfası'
      on Click: ActivateScreen("Reçete", 0)
*)